Fanuc KAREL source: kt00182.KL

-- PROVISIONAL review KL for V940-1; original PC SHA256 799ae98dc465ca07837d44aa42971392e01c9ef045778bfb8728f611b592f2c1
-- Incomplete behavior may be omitted. Consult companion uncertainty JSON. Do not deploy.
PROGRAM KT00182
%NOLOCKGROUP
VAR
  OUT : REAL
-- UNRESOLVED_DECL Y1 type=002018
-- UNRESOLVED_DECL Y2 type=002018
BEGIN
  -- V9_ZERO_TABLE_METADATA_HINT layout=0001; no indexed target words; source/name/runtime held
  -- UNRESOLVED_PC offsets 5-19; opcodes 2E,22,9D,33,B2
  -- UNRESOLVED_PC offsets 24-38; opcodes 2E,22,9D,33,B2
  -- UNRESOLVED_PC offsets 43-57; opcodes 2E,22,9D,33,B2
  -- UNRESOLVED_PC offsets 62-76; opcodes 2E,22,9D,33,B2
  -- UNRESOLVED_PC offsets 81-107; opcodes 22,9D,33,B1,22,9D,33,B1,56,64,23
  -- UNRESOLVED_PC offsets 112-116; opcodes 7F
END KT00182
